// TIA Portal V18 export
// export: Created 2026-06-08T16:08:49.8901737Z, ExportSetting WithDefaults, DisplayName Totally Integrated Automation Portal, DisplayVersion V18, DisplayName TIA Portal Openness, DisplayVersion V18, DisplayName TIA Portal Version Control Interface, DisplayVersion V18, DisplayName STEP 7 Professional, DisplayVersion V18, DisplayName STEP 7 Safety, DisplayVersion V18, DisplayName WinCC Professional, DisplayVersion V18
ORGANIZATION_BLOCK "Main"   // OB1, LAD, ProgramCycle
TITLE = "Main Program Sweep (Cycle)"
{ S7_Optimized_Access := 'TRUE' }
VERSION : 0.1
// stored: AutoNumber true, IsIECCheckEnabled false, SetENOAutomatically false
   VAR_INPUT
      Initial_Call : Bool;   // Initial call of this OB
      Remanence : Bool;   // =True, if remanent data are available
   END_VAR
   VAR_TEMP
      TG_ND : Int;
      TG_ND1 : Real;
   END_VAR
BEGIN

REGION Network 1: Điều khiển đèn làm việc
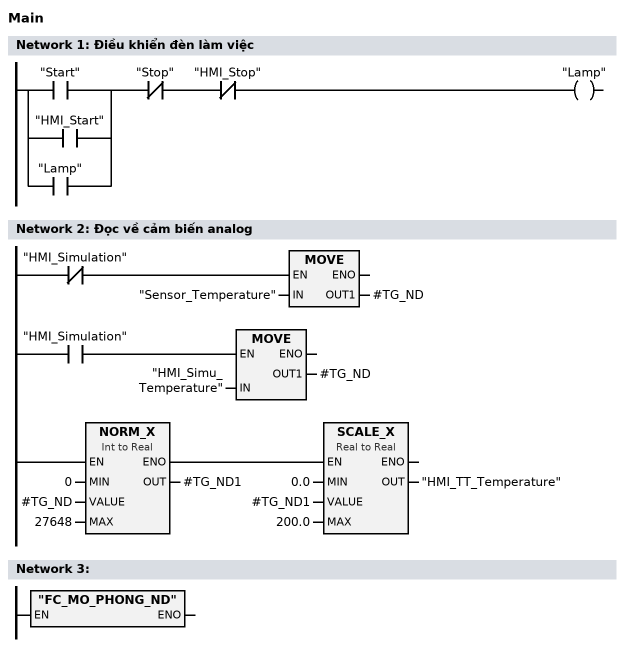
   RUNG wire#powerrail
      Contact( "Start" )
      wire#w1
      I_Contact( "Stop" )
      I_Contact( "HMI_Stop" )
      Coil( "Lamp" )
   END_RUNG
   RUNG wire#powerrail
      Contact( "HMI_Start" )
   END_RUNG wire#w1
   RUNG wire#powerrail
      Contact( "Lamp" )
   END_RUNG wire#w1
   // the same network as SCL:
   "Lamp" := ("Start" OR "HMI_Start" OR "Lamp") AND NOT "Stop" AND NOT "HMI_Stop";
END_REGION

REGION Network 2: Đọc về cảm biến analog
   RUNG wire#powerrail
      I_Contact( "HMI_Simulation" )
      Move(in := "Sensor_Temperature", out1 => #TG_ND)
   END_RUNG
   RUNG wire#powerrail
      Contact( "HMI_Simulation" )
      Move(in := "HMI_Simu_Temperature", out1 => #TG_ND)
   END_RUNG
   RUNG wire#powerrail
      { S7_Templates := "[SrcType := Int, DestType := Real]" } Normalize(min := 0, value := #TG_ND, max := 27648, out => #TG_ND1)
      { S7_Templates := "[SrcType := Real, DestType := Real]" } Scale(min := 0.0, value := #TG_ND1, max := 200.0, out => "HMI_TT_Temperature")
   END_RUNG
   // the same network as SCL:
   IF NOT "HMI_Simulation" THEN #TG_ND := "Sensor_Temperature"; END_IF;
   IF "HMI_Simulation" THEN #TG_ND := "HMI_Simu_Temperature"; END_IF;
   #TG_ND1 := NORM_X(MIN := 0, VALUE := #TG_ND, MAX := 27648);
   "HMI_TT_Temperature" := SCALE_X(MIN := 0.0, VALUE := #TG_ND1, MAX := 200.0);
END_REGION

REGION Network 3
   RUNG wire#powerrail
      "FC_MO_PHONG_ND"()
   END_RUNG
   // the same network as SCL:
   "FC_MO_PHONG_ND"();
END_REGION
END_ORGANIZATION_BLOCK
